FUNCTION SPLITTING_WORD_TO_QUARTERS
  (* Standard: 61499-1; Description: Copyright (c) 2024 HR Agrartechnik GmbH This program and the accompanying materials are made available under the terms of the Eclipse Public License 2.0 which is available at https://www.eclipse.org/legal/epl-2.0/ SPDX-License-Identifier: EPL-2.0 *)
  (* Version 1.0, 2024-02-22, franz *)
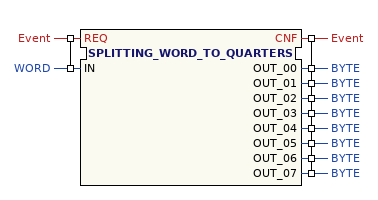
  EVENT_INPUT
    REQ WITH IN; (* Normal Execution Request *)
  END_EVENT
  EVENT_OUTPUT
    CNF WITH OUT_00, OUT_01, OUT_02, OUT_03, OUT_04, OUT_05, OUT_06, OUT_07; (* Execution Confirmation *)
  END_EVENT
  VAR_INPUT
    IN : WORD; (* WORD Input *)
  END_VAR
  VAR_OUTPUT
    OUT_00 : BYTE; (* QUARTER BYTE 00 *)
    OUT_01 : BYTE; (* QUARTER BYTE 01 *)
    OUT_02 : BYTE; (* QUARTER BYTE 02 *)
    OUT_03 : BYTE; (* QUARTER BYTE 03 *)
    OUT_04 : BYTE; (* QUARTER BYTE 04 *)
    OUT_05 : BYTE; (* QUARTER BYTE 05 *)
    OUT_06 : BYTE; (* QUARTER BYTE 06 *)
    OUT_07 : BYTE; (* QUARTER BYTE 07 *)
  END_VAR
  BODY IN ST:
FUNCTION SPLITTING_WORD_TO_QUARTERS

VAR_INPUT
	IN : WORD;    // WORD Input
END_VAR

VAR_OUTPUT
	OUT_00 : BYTE;    // QUARTER BYTE 00
	OUT_01 : BYTE;    // QUARTER BYTE 01
	OUT_02 : BYTE;    // QUARTER BYTE 02
	OUT_03 : BYTE;    // QUARTER BYTE 03
	OUT_04 : BYTE;    // QUARTER BYTE 04
	OUT_05 : BYTE;    // QUARTER BYTE 05
	OUT_06 : BYTE;    // QUARTER BYTE 06
	OUT_07 : BYTE;    // QUARTER BYTE 07
END_VAR

(* this Function extracts the 8 QUARTER BYTE from a word *)
OUT_00 := WORD_TO_BYTE(SHR(IN AND WORD_QUARTER_00, SHFT_QUARTER_00));
OUT_01 := WORD_TO_BYTE(SHR(IN AND WORD_QUARTER_01, SHFT_QUARTER_01));
OUT_02 := WORD_TO_BYTE(SHR(IN AND WORD_QUARTER_02, SHFT_QUARTER_02));
OUT_03 := WORD_TO_BYTE(SHR(IN AND WORD_QUARTER_03, SHFT_QUARTER_03));
OUT_04 := WORD_TO_BYTE(SHR(IN AND WORD_QUARTER_04, SHFT_QUARTER_04));
OUT_05 := WORD_TO_BYTE(SHR(IN AND WORD_QUARTER_05, SHFT_QUARTER_05));
OUT_06 := WORD_TO_BYTE(SHR(IN AND WORD_QUARTER_06, SHFT_QUARTER_06));
OUT_07 := WORD_TO_BYTE(SHR(IN AND WORD_QUARTER_07, SHFT_QUARTER_07));

END_FUNCTION
  END_BODY
END_FUNCTION
